# EPICS substitutions: apps/amqApp/Db/amqTriggerBits.substitutions
file "db/amqDouble.db" {
    pattern { P K THH TH HHSV HSV EGU }
    { B_DAQ:livetime TRIG1_TSLIVETIMESLOT21 10 20 MINOR MAJOR "%" }
    { B_DAQ:PRAD:livetime TRIG0_TSLIVETIMESLOT21 10 20 MINOR MAJOR "%" }
}

file "db/amqTrigBit.template" {
    pattern { INOPT N M DESC }
    { "CPP"  0  1 "Electron - OR of 1-6" }
    { ""     1  2 "S1" }
    { ""     2  3 "S2" }
    { ""     3  4 "S3" }
    { ""     4  5 "S4" }
    { ""     5  6 "S5" }
    { ""     6  7 "S6" }
    { ""     7  8 "HTCC1" }
    { ""     8  9 "HTCC2" }
    { ""     9 10 "HTCC3" }
    { ""    10 11 "HTCC4" }
    { ""    11 12 "HTCC5" }
    { ""    12 13 "HTCC6" }
    { ""    13 14 "PCAL1" }
    { ""    14 15 "PCAL2" }
    { ""    15 16 "PCAL3" }
    { ""    16 17 "PCAL4" }
    { ""    17 18 "PCAL5" }
    { ""    18 19 "PCAL6" }
    { ""    19 20 "ECAL1" }
    { ""    20 21 "ECAL2" }
    { ""    21 22 "ECAL3" }
    { ""    22 23 "ECAL4" }
    { ""    23 24 "ECAL5" }
    { ""    24 25 "ECAL6" }
    { ""    25 26 "HTCC x PCAL>60MeV" }
    { ""    26 27 "HTCC x PCAL>150MeV" }
    { ""    27 28 "PCAL x ECAL" }
    { ""    28 29 "FTOF x PCAL" }
    { ""    29 30 "FTC > 10 MeV" }
    { ""    30 31 "FTC > 50 MeV" }
    { ""    31 32 "Pulser" }
}

file "db/amqTrig-TS.template" {
    pattern { INOPT N M DESC }
    { "CPP" 0 1 0 }
    { ""    1 2 1 }
    { ""    2 3 2 }
    { ""    3 4 3 }
    { ""    4 5 4 }
    { ""    5 6 5 }
    { ""    6 7 6 }
    { ""    7 8 7 }
    { ""    8 9 8 }
    { ""    9 10 9 }
    { ""    10 11 10 }
    { ""    11 12 11 }
    { ""    12 13 12 }
    { ""    13 14 13 }
    { ""    14 15 14 }
    { ""    15 16 15 }
    { ""    16 17 16 }
    { ""    17 18 17 }
    { ""    18 19 18 }
    { ""    19 20 19 }
    { ""    20 21 20 }
    { ""    21 22 21 }
    { ""    22 23 22 }
    { ""    23 24 23 }
    { ""    24 25 24 }
    { ""    25 26 25 }
    { ""    26 27 26 }
    { ""    27 28 27 }
    { ""    28 29 28 }
    { ""    29 30 29 }
    { ""    30 31 30 }
    { ""    31 32 31 }
}

file "db/amqTrigBit-stage2.template" { pattern { S } { 1 } { 2 } { 3 } { 4 } { 5 } { 6 } }

file "db/amqDoubleArray.db" {
pattern { P K N TH THH HSV HHSV }
    { B_DAQ:dc11vtp_VTPDC_SUPERLAYER dc11vtp_VTPDC_SUPERLAYER 6 10 20 MINOR MAJOR }
    { B_DAQ:dc12vtp_VTPDC_SUPERLAYER dc12vtp_VTPDC_SUPERLAYER 6 10 20 MINOR MAJOR }
    { B_DAQ:dc13vtp_VTPDC_SUPERLAYER dc13vtp_VTPDC_SUPERLAYER 6 10 20 MINOR MAJOR }

    { B_DAQ:dc21vtp_VTPDC_SUPERLAYER dc21vtp_VTPDC_SUPERLAYER 6 10 20 MINOR MAJOR }
    { B_DAQ:dc22vtp_VTPDC_SUPERLAYER dc22vtp_VTPDC_SUPERLAYER 6 10 20 MINOR MAJOR }
    { B_DAQ:dc23vtp_VTPDC_SUPERLAYER dc23vtp_VTPDC_SUPERLAYER 6 10 20 MINOR MAJOR }

    { B_DAQ:dc31vtp_VTPDC_SUPERLAYER dc31vtp_VTPDC_SUPERLAYER 6 10 20 MINOR MAJOR }
    { B_DAQ:dc32vtp_VTPDC_SUPERLAYER dc32vtp_VTPDC_SUPERLAYER 6 10 20 MINOR MAJOR }
    { B_DAQ:dc33vtp_VTPDC_SUPERLAYER dc33vtp_VTPDC_SUPERLAYER 6 10 20 MINOR MAJOR }

    { B_DAQ:dc41vtp_VTPDC_SUPERLAYER dc41vtp_VTPDC_SUPERLAYER 6 10 20 MINOR MAJOR }
    { B_DAQ:dc42vtp_VTPDC_SUPERLAYER dc42vtp_VTPDC_SUPERLAYER 6 10 20 MINOR MAJOR }
    { B_DAQ:dc43vtp_VTPDC_SUPERLAYER dc43vtp_VTPDC_SUPERLAYER 6 10 20 MINOR MAJOR }

    { B_DAQ:dc51vtp_VTPDC_SUPERLAYER dc51vtp_VTPDC_SUPERLAYER 6 10 20 MINOR MAJOR }
    { B_DAQ:dc52vtp_VTPDC_SUPERLAYER dc52vtp_VTPDC_SUPERLAYER 6 10 20 MINOR MAJOR }
    { B_DAQ:dc53vtp_VTPDC_SUPERLAYER dc53vtp_VTPDC_SUPERLAYER 6 10 20 MINOR MAJOR }

    { B_DAQ:dc61vtp_VTPDC_SUPERLAYER dc61vtp_VTPDC_SUPERLAYER 6 10 20 MINOR MAJOR }
    { B_DAQ:dc62vtp_VTPDC_SUPERLAYER dc62vtp_VTPDC_SUPERLAYER 6 10 20 MINOR MAJOR }
    { B_DAQ:dc63vtp_VTPDC_SUPERLAYER dc63vtp_VTPDC_SUPERLAYER 6 10 20 MINOR MAJOR }

    { B_DAQ:dc11vtp_VTPDC_SUPERLAYER dc11vtp_VTPDC_SUPERLAYER 6 10 20 MINOR MAJOR }
    { B_DAQ:dc12vtp_VTPDC_SUPERLAYER dc12vtp_VTPDC_SUPERLAYER 6 10 20 MINOR MAJOR }
    { B_DAQ:dc13vtp_VTPDC_SUPERLAYER dc13vtp_VTPDC_SUPERLAYER 6 10 20 MINOR MAJOR }
}

file "db/amqDoubleArray.db" {
pattern { P K N TH THH HSV HHSV }
{    SSPGTC_SLOT9_FTCLUSTER_RATE          SSPGTC_SLOT9_FTCLUSTER_RATE 2 10 20 MINOR MAJOR }
{    SSPGTC_SLOT10_FTCLUSTER_RATE         SSPGTC_SLOT10_FTCLUSTER_RATE 2 10 20 MINOR MAJOR }
{    adcft1vtp_VTPFT_HODOSCALERS          adcft1vtp_VTPFT_HODOSCALERS 256 10 20 MINOR MAJOR }
{    adcft1vtp_VTPFT_CLUSTERPOSITION      adcft1vtp_VTPFT_CLUSTERPOSITION 1024 10 20 MINOR MAJOR }
{    adcft1vtp_VTPFT_CLUSTERENERGY        adcft1vtp_VTPFT_CLUSTERENERGY 1024 10 20 MINOR MAJOR }
{    adcft1vtp_VTPFT_CLUSTERHITS          adcft1vtp_VTPFT_CLUSTERHITS 9 10 20 MINOR MAJOR }
{    adcft1vtp_VTPFT_CLUSTERPOSITION_HODO adcft1vtp_VTPFT_CLUSTERPOSITION_HODO 1024 10 20 MINOR MAJOR }
{    adcft1vtp_VTPFT_CLUSTERENERGY_HODO   adcft1vtp_VTPFT_CLUSTERENERGY_HODO 1024 10 20 MINOR MAJOR }
{    adcft1vtp_VTPFT_CLUSTERNHITS_HODO    adcft1vtp_VTPFT_CLUSTERNHITS_HODO 9 10 20 MINOR MAJOR }
{    adcft2vtp_VTPFT_HODOSCALERS          adcft2vtp_VTPFT_HODOSCALERS 256 10 20 MINOR MAJOR }
{    adcft2vtp_VTPFT_CLUSTERPOSITION      adcft2vtp_VTPFT_CLUSTERPOSITION 1024 10 20 MINOR MAJOR }
{    adcft2vtp_VTPFT_CLUSTERENERGY        adcft2vtp_VTPFT_CLUSTERENERGY 1024 10 20 MINOR MAJOR }
{    adcft2vtp_VTPFT_CLUSTERHITS          adcft2vtp_VTPFT_CLUSTERHITS 9 10 20 MINOR MAJOR }
{    adcft2vtp_VTPFT_CLUSTERPOSITION_HODO adcft2vtp_VTPFT_CLUSTERPOSITION_HODO 1024 10 20 MINOR MAJOR }
{    adcft2vtp_VTPFT_CLUSTERENERGY_HODO   adcft2vtp_VTPFT_CLUSTERENERGY_HODO 1024 10 20 MINOR MAJOR }
{    adcft2vtp_VTPFT_CLUSTERNHITS_HODO    adcft2vtp_VTPFT_CLUSTERNHITS_HODO 9 10 20 MINOR MAJOR }
{    adcft3vtp_VTPFT_HODOSCALERS          adcft3vtp_VTPFT_HODOSCALERS 256 10 20 MINOR MAJOR }
{    adcft3vtp_VTPFT_CLUSTERPOSITION      adcft3vtp_VTPFT_CLUSTERPOSITION 1024 10 20 MINOR MAJOR }
{    adcft3vtp_VTPFT_CLUSTERENERGY        adcft3vtp_VTPFT_CLUSTERENERGY 1024 10 20 MINOR MAJOR }
{    adcft3vtp_VTPFT_CLUSTERHITS          adcft3vtp_VTPFT_CLUSTERHITS 9 10 20 MINOR MAJOR }
{    adcft3vtp_VTPFT_CLUSTERPOSITION_HODO adcft3vtp_VTPFT_CLUSTERPOSITION_HODO 1024 10 20 MINOR MAJOR }
{    adcft3vtp_VTPFT_CLUSTERENERGY_HODO   adcft3vtp_VTPFT_CLUSTERENERGY_HODO 1024 10 20 MINOR MAJOR }
{    adcft3vtp_VTPFT_CLUSTERNHITS_HODO    adcft3vtp_VTPFT_CLUSTERNHITS_HODO 9 10 20 MINOR MAJOR }
}

file "db/amqMergeFT.db" {
pattern { IN1 IN2 P N }
{    adcft1vtp_VTPFT_HODOSCALERS          adcft2vtp_VTPFT_HODOSCALERS          VTPFT_HODOSCALERS 256 }
{    adcft1vtp_VTPFT_CLUSTERPOSITION      adcft2vtp_VTPFT_CLUSTERPOSITION      VTPFT_CLUSTERPOSITION 1024 }
{    adcft1vtp_VTPFT_CLUSTERENERGY        adcft2vtp_VTPFT_CLUSTERENERGY        VTPFT_CLUSTERENERGY 1024 }
{    adcft1vtp_VTPFT_CLUSTERHITS          adcft2vtp_VTPFT_CLUSTERHITS          VTPFT_CLUSTERHITS 9 }
{    adcft1vtp_VTPFT_CLUSTERPOSITION_HODO adcft2vtp_VTPFT_CLUSTERPOSITION_HODO VTPFT_CLUSTERPOSITION_HODO 1024 }
{    adcft1vtp_VTPFT_CLUSTERENERGY_HODO   adcft2vtp_VTPFT_CLUSTERENERGY_HODO   VTPFT_CLUSTERENERGY_HODO 1024 }
{    adcft1vtp_VTPFT_CLUSTERNHITS_HODO    adcft2vtp_VTPFT_CLUSTERNHITS_HODO    VTPFT_CLUSTERNHITS_HODO 9 }
}

file "db/amqDoubleArray.db" {
pattern { P K N TH THH HSV HHSV }
{ B_DAQ:trig2vtp_VTPGT_PRESCALES   trig2vtp_VTPGT_PRESCALES   32 0 30 NO_ALARM MAJOR }
{ B_DAQ:trig1ts_TRIGGERBITS        TRIG1_TSGTPSLOT21          32 0 30 NO_ALARM MAJOR }
{ B_DAQ:trig1tsfp_TRIGGERBITS      TRIG1_TSFPSLOT21           32 0 30 NO_ALARM MAJOR }
{ B_DAQ:trig1tsfp_PRESCALES        TRIG1_TSFPPRESCALESSLOT21  32 0 30 NO_ALARM MAJOR }
{ B_DAQ:trig1ts_PRESCALES          TRIG1_TSGTPPRESCALESSLOT21 32 0 30 NO_ALARM MAJOR }
}

file "db/array-to-scalar-32.template" {
pattern { P R S INP FTVL }
{ B_DAQ:trig2vtp_VTPGT_PRESCALES:  "" "" B_DAQ:trig2vtp_VTPGT_PRESCALES FLOAT }
{ B_DAQ:trig1ts_TRIGGERBITS:       "" "" B_DAQ:trig1ts_TRIGGERBITS      FLOAT }
{ B_DAQ:trig1tsfp_TRIGGERBITS:     "" "" B_DAQ:trig1tsfp_TRIGGERBITS    FLOAT }
{ B_DAQ:trig1tsfp_PRESCALES:       "" "" B_DAQ:trig1tsfp_PRESCALES      FLOAT }
{ B_DAQ:trig1ts_PRESCALES:         "" "" B_DAQ:trig1ts_PRESCALES        FLOAT }
}

file "db/amqTrigFrac.template" {
pattern { P BIT BIT2 }
{ B_DAQ:trig1ts_TRIGGERBITS 0 00 }
{ B_DAQ:trig1ts_TRIGGERBITS 1 01 }
{ B_DAQ:trig1ts_TRIGGERBITS 2 02 }
{ B_DAQ:trig1ts_TRIGGERBITS 3 03 }
{ B_DAQ:trig1ts_TRIGGERBITS 4 04 }
{ B_DAQ:trig1ts_TRIGGERBITS 5 05 }
{ B_DAQ:trig1ts_TRIGGERBITS 6 06 }
{ B_DAQ:trig1ts_TRIGGERBITS 7 07 }
{ B_DAQ:trig1ts_TRIGGERBITS 8 08 }
{ B_DAQ:trig1ts_TRIGGERBITS 9 09 }
{ B_DAQ:trig1ts_TRIGGERBITS 10 10 }
{ B_DAQ:trig1ts_TRIGGERBITS 11 11 }
{ B_DAQ:trig1ts_TRIGGERBITS 12 12 }
{ B_DAQ:trig1ts_TRIGGERBITS 13 13 }
{ B_DAQ:trig1ts_TRIGGERBITS 14 14 }
{ B_DAQ:trig1ts_TRIGGERBITS 15 15 }
{ B_DAQ:trig1ts_TRIGGERBITS 16 16 }
{ B_DAQ:trig1ts_TRIGGERBITS 17 17 }
{ B_DAQ:trig1ts_TRIGGERBITS 18 18 }
{ B_DAQ:trig1ts_TRIGGERBITS 19 19 }
{ B_DAQ:trig1ts_TRIGGERBITS 20 20 }
{ B_DAQ:trig1ts_TRIGGERBITS 21 21 }
{ B_DAQ:trig1ts_TRIGGERBITS 22 22 }
{ B_DAQ:trig1ts_TRIGGERBITS 23 23 }
{ B_DAQ:trig1ts_TRIGGERBITS 24 24 }
{ B_DAQ:trig1ts_TRIGGERBITS 25 25 }
{ B_DAQ:trig1ts_TRIGGERBITS 26 26 }
{ B_DAQ:trig1ts_TRIGGERBITS 27 27 }
{ B_DAQ:trig1ts_TRIGGERBITS 28 28 }
{ B_DAQ:trig1ts_TRIGGERBITS 29 29 }
{ B_DAQ:trig1ts_TRIGGERBITS 30 30 }
{ B_DAQ:trig1ts_TRIGGERBITS 31 31 }
}
